{attribute 'no_explicit_call' := 'do not call this POU directly'} 
// Provide the functionality to use more than one Logger target
FUNCTION_BLOCK FB_LoggerManager IMPLEMENTS I_Logger
VAR
	nLength:		INT;
	pList: 			POINTER TO I_Logger;
	aList:			POINTER TO POINTER TO ARRAY [0..24] OF I_Logger:=ADR(pList);
END_VAR

// https://peterzerlauth.com/

METHOD FB_exit : BOOL
VAR_INPUT
	bInCopyCode : BOOL; // if TRUE, the exit method is called for exiting an instance that is copied afterwards (online change).
END_VAR
M_Clear();
END_METHOD

METHOD PUBLIC M_Add : BOOL
VAR_INPUT
	iLogger: 	I_Logger;
END_VAR
VAR
	pOldList: 	POINTER TO I_Logger;
END_VAR
IF iLogger <> 0 THEN
	// First Item
	IF pList = 0 THEN
		nLength:= nLength + 1;
		pList:= __NEW(POINTER TO I_Logger, DINT_TO_UDINT(nLength));
	ELSE
		// Item already in List
		IF M_Find(iLogger) = -1 THEN
			// backup 
			pOldList:= pList;
			// new Length
			nLength:= nLength + 1;
			// new pointer
			pList:= __NEW(POINTER TO I_Logger, DINT_TO_UDINT(nLength));
			// restore
			Memcpy(pList, pOldList, SIZEOF(pList) * DINT_TO_UDINT(nLength -1));
			// delete old
			__DELETE(pOldList);
		ELSE
			M_Add:= FALSE;	
			RETURN;
		END_IF
	END_IF
	IF pList = 0 THEN
		RETURN;
	END_IF
	// add new Object
	pList[nLength-1]:= iLogger;
	M_Add:= TRUE;
ELSE
	M_Add:= FALSE;	
END_IF
END_METHOD

METHOD PUBLIC M_Clear : bool
IF pList <> 0 THEN
	nLength:= 0;
	__DELETE(pList);
END_IF
M_Clear:= TRUE;
END_METHOD

METHOD PUBLIC M_Find : DINT
VAR_INPUT
	iLogger: 	I_Logger;
END_VAR
VAR
	nIndex: 	UINT;
END_VAR
// Object already in List
M_Find := -1;
WHILE nIndex < nLength DO
    IF (pList[nIndex] = iLogger) THEN
        M_Find := nIndex;
        RETURN;
    END_IF
	nIndex := nIndex + 1;
END_WHILE
END_METHOD

METHOD PUBLIC M_Index : I_Logger
VAR_INPUT
	nIndex: 	DINT;
END_VAR
IF (nIndex < nLength) THEN
	M_Index := pList[nIndex];
END_IF
END_METHOD

METHOD PUBLIC M_Log : BOOL
VAR_INPUT
	fbMessage:			FB_Message;
END_VAR
VAR
	nIndex:		INT;
END_VAR
WHILE nIndex < nLength DO
    pList[nIndex].M_Log(fbMessage);
	nIndex := nIndex + 1;
END_WHILE
END_METHOD

METHOD PUBLIC M_Remove : BOOL
VAR_INPUT
	iLogger: 	I_Logger;
END_VAR
VAR
	pOldList:			POINTER TO I_Logger;
	nPosition: 			DINT;
END_VAR
IF iLogger <> 0 THEN
	// First Item
	IF nLength >= 0 THEN
		// Item already in List
		nPosition:= M_Find(iLogger);
		IF nPosition <> -1 THEN
			// backup 
			pOldList:= pList;
			// new Length
			nLength:= nLength -1;
			// new pointer
			pList:= __NEW(POINTER TO I_Logger ,DINT_TO_UDINT(nLength));
			// restore lower part
			Memcpy(pList, pOldList, SIZEOF(pList) * DINT_TO_UDINT(nPosition));
			//pList[nPosition]:= iObject;
			Memcpy(pList + (SIZEOF(pList) * nPosition),pOldList + (SIZEOF(pList)*(nPosition + 1)), SIZEOF(pList) * DINT_TO_UDINT(nLength - nPosition));
			// delete old
			__DELETE(pOldList);
		ELSE
			M_Remove:= FALSE;	
			RETURN;
		END_IF
	ELSE
		M_Remove:= FALSE;	
		RETURN;
	END_IF
	M_Remove:= TRUE;
ELSE
	M_Remove:= FALSE;	
END_IF
END_METHOD

METHOD M_Reset : BOOL
VAR_INPUT
END_VAR
VAR
	nIndex: 				UINT;
END_VAR
nIndex := 0;
WHILE nIndex < nLength DO
    pList[nIndex].M_Reset();
    nIndex := nIndex + 1;
END_WHILE
M_Reset:= TRUE;
END_METHOD

{attribute 'OPC.UA.DA.Property' := '1'}
{attribute 'monitoring' := 'variable'}
PROPERTY PUBLIC P_Length : INT
GET
P_Length:= nLength;
END_GET
END_PROPERTY

END_FUNCTION_BLOCK

(* stored: Version 1.1.0.1
   POU FB_LoggerManager: Id {8d6eb986-1a4b-011f-072f-86ab56dd3ee8}, SpecialFunc None
   Method FB_exit: Id {f2cbd9f6-7524-0c7f-39f0-dce225abbc0c}
   Method M_Add: Id {48be3447-76e8-0bc8-0db5-61654f9fc9a9}
   Method M_Clear: Id {8b758e8a-4901-0f32-3045-a207842a9e60}
   Method M_Find: Id {37f499ab-a90c-0435-0594-f330a6c37cb8}
   Method M_Index: Id {c0986c64-83e2-03be-09c2-3f0e829e981d}
   Method M_Log: Id {179441ef-3445-0ab5-3cfb-99e937e75dd0}
   Method M_Remove: Id {344ce544-0b6b-0e0a-1940-689d2bdbdc8d}
   Method M_Reset: Id {1ef4ca52-3820-45a5-a9c2-ebd6113db930}
   Property P_Length: Id {cf1d82fc-0cbb-0b4a-372a-308b43a41775}
   Get Get: Id {378639c8-9631-0870-37c8-2847124df936} *)
